{library PUBLIC}
(* Function to start a assembly process on the table. *)
FUNCTION_BLOCK ABBProcessAssembly
VAR_INPUT
	En: 				BOOL:=FALSE;			(* Set to true to start *)
END_VAR
VAR_OUTPUT
	Done: 				BOOL:=FALSE;			(* If true, the command is transmitted ok, to reset set En to false *)
	Executing:			BOOL:=FALSE;			(* True while the command in transmitted *)
	Waiting:			BOOL:=FALSE;			(* True if the command is queued to be transmitted *)
	Error: 				BOOL := FALSE;			(* True if an error occured *)
	Progress:			INT:=0;						(* Function progress *)
END_VAR
VAR_IN_OUT
	Data: 				CommunicationData;		(* Common data structure to connect this function block to a specific Communicator block *)
END_VAR
VAR
	FunctionType: 		FUNCTION_TYPE;
	FunctionNumber: 	INT;
	ParameterDW:	DWORD;
	ParameterB:		BYTE;
	Sequence:			INT:=0;

	fbRPC:				ASyncRPC;
END_VAR

FunctionType:=FUNCTION_TYPE.FUNCTION_TYPE_ASYNC_RPC;
FunctionNumber:=ABB_ASYNC_FUNCTION_PROCESS_ASSEMBLY;
ParameterDW:=0;
ParameterB:=0;

fbRPC(EN:=En, Data:=Data, FunctionType:=FunctionType,FunctionNumber:=FunctionNumber, ParameterDW:=ParameterDW, ParameterB:=ParameterB);

Done:=fbRPC.Done;
Executing:=fbRPC.Executing;
Waiting:=fbRPC.Waiting;
Error:=fbRPC.Error OR (fbRPC.Done AND fbRPC.ReturnValue<0);
Progress:=fbRPC.Progress;

END_FUNCTION_BLOCK

(* stored: Version 1.1.0.1, ProductVersion 3.1.4022.12
   POU ABBProcessAssembly: Id {4a63d37d-7c98-4c33-a3ce-b3e7983ab354}, SpecialFunc None *)
